RoboDK station: UR3e simulation_test1.rdk

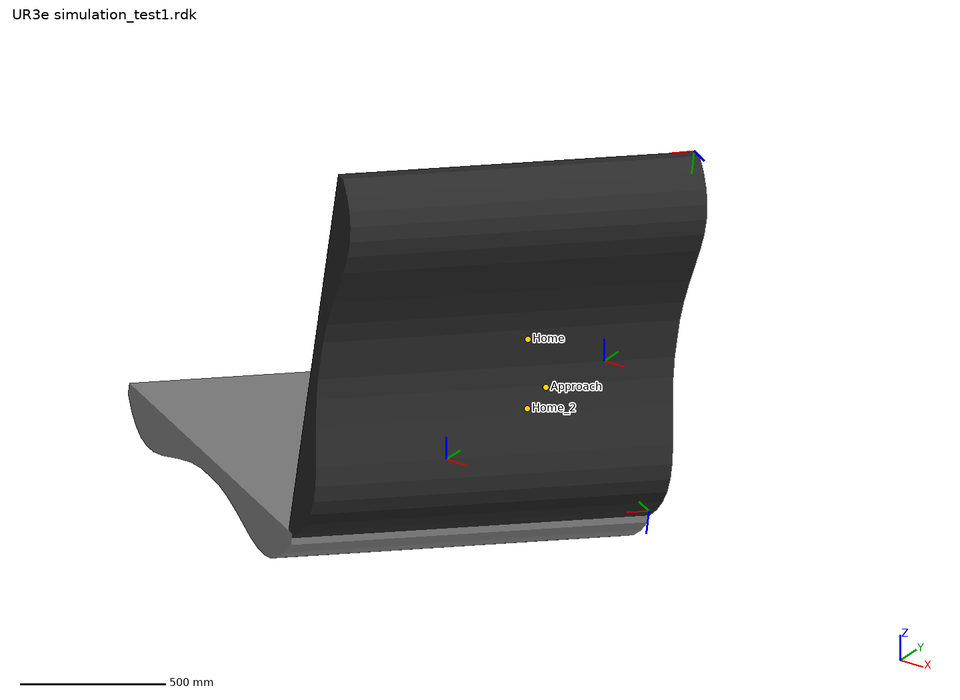
[picture v0: the station drawn from its stored meshes, robots at their saved joint values, targets as dots, program paths as lines]
Station UR3e simulation_test1 (saved by RoboDK 5.8.0). Poses are relative to the parent item; angles as X-Y-Z fixed-axis rotations.
  - frame UR3e Base at (0, 14.75, 0) mm, rotated rx 0 ry -0.13 rz 0 deg
    - robot UR3e: 6 axes, payload 3 kg, reach 500 mm, repeatability 0.03 mm, weight 11 kg
        modified DH rows (alpha deg, a mm, theta deg, d mm): 0, 0, 0, 151.9; 90, 0, 180, 0; 0, 243.55, 0, 0; 0, 213.2, 0, 131.05; -90, 0, 0, 85.35; 90, 0, 180, 92.1
        joint limits [-360, -360, -360, -360, -360, -360] to [360, 360, 360, 360, 360, 360]; home [0, -90, -90, 0, 90, 0]; saved at [-34.234, -79.814, -98.873, 0.742, 174.902, 2.275]
      - tool Paint gun, TCP at (-49.23, 0, 278.13) mm, rotated rx 0 ry 30 rz 0 deg, size 203.2 x 279.7 x 471.5 mm
    - frame Frame 2 at (0, 942.71, 0) mm
      - target Home_2 (Cartesian target) at (394.25, -1020.68, 334.7) mm, rotated rx -105.88 ry 0 rz -120 deg; joints [-2.778, -38.293, -133.63, -21.811, 93.645, 7.204] of UR3e
      - target Approach (Cartesian target) at (523.34, -1095.21, 480.8) mm, rotated rx -90 ry 0 rz -120 deg; joints [-21.639, -90.825, -89.168, -0.007, 111.639, 0] of UR3e
      - target Home (Cartesian target) at (260.91, -827.44, 483.17) mm, rotated rx -89.96 ry 0.29 rz -69.33 deg; joints [-34.234, -79.814, -98.873, 0.742, 174.902, 2.275] of UR3e
  - Python program Paint_hexagonalmove (listed below)
  - frame Frame 3 at (740.28, 167.78, -52.56) mm, rotated rx -178.96 ry -7.72 rz -120.73 deg
    - object Object Inspection at (0, 0, 0) mm, size 1355.2 x 1355.2 x 156.4 mm, geometry from Object Inspection.stp
  - frame Frame 4 at (817.38, 331.94, 1278.48) mm, rotated rx -90.65 ry -7.72 rz -120.73 deg
    - object Object Inspection at (0, 0, 0) mm, size 1355.2 x 1355.2 x 156.4 mm, geometry from Object Inspection.stp

--- Python program Paint_hexagonalmove ---
from robolink import *    # API to communicate with RoboDK
from robodk import *      # robodk robotics toolbox

# Any interaction with RoboDK must be done through RDK:
RDK = Robolink()

# get the robot by name:
robot = RDK.Item('', ITEM_TYPE_ROBOT)

# get the home target and the welding targets:
home = RDK.Item('Home')
target = RDK.Item('Approach')

# get the pose of the target (4x4 matrix representing position and orientation):
poseref = target.Pose()

# move the robot to home, then to the Target 1:
robot.MoveJ(home)
robot.MoveJ(target)

# make an hexagon around the Target 1:
for i in range(7):
    ang = i*2*pi/6 #angle: 0, 60, 120, ...
    posei = poseref*rotz(ang)*transl(130,0,0)*rotz(-ang)
    robot.MoveL(posei)

# move back to the center, then home:
robot.MoveL(target)
robot.MoveJ(home)
